RoboDK station: ICGI2018_station.rdk

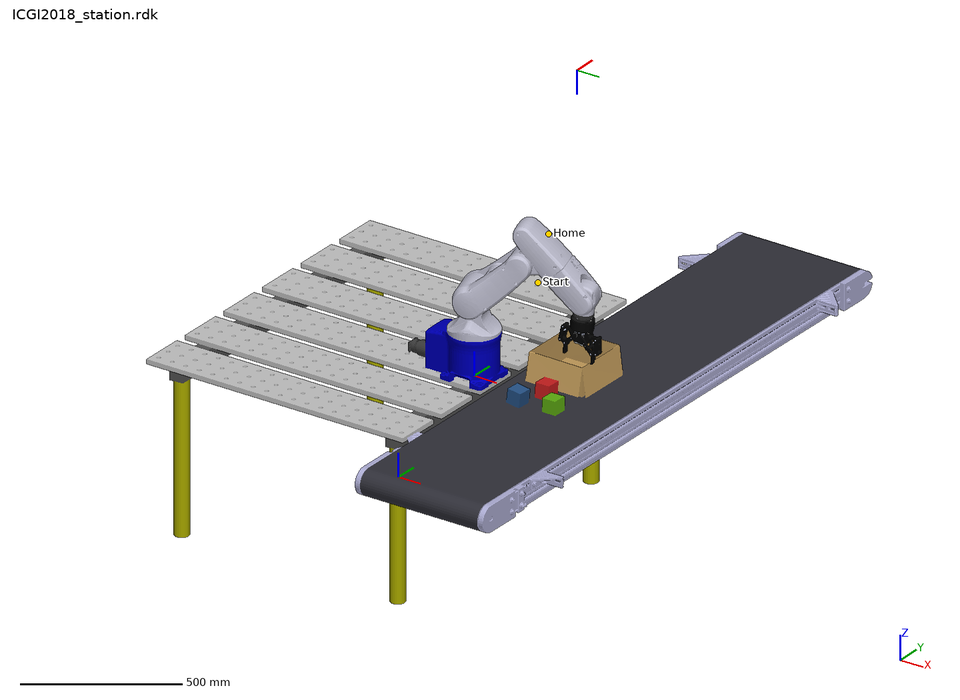
[picture v0: the station drawn from its stored meshes, robots at their saved joint values, targets as dots, program paths as lines]
Station ICGI2018_station. Poses are relative to the parent item; angles as X-Y-Z fixed-axis rotations.
  - frame ConveyorReference at (216.46, -62.53, 0) mm
    - object Conveyor at (-115.17, 300, -50) mm, size 597 x 2090.8 x 107.2 mm
    - object Opened Box at (-58.27, 786.37, -1) mm, size 224.8 x 231.5 x 101.8 mm, geometry from box.stl
  - object Object Table at (-409.94, 767.55, 0) mm, rotated rx 0 ry 0 rz -90.17 deg, size 1193.8 x 965.2 x 609.6 mm, geometry from Object Table.wrl
  - program ResetPositions (1 instructions, listed below)
  - frame Camera Frame at (325.51, 738.58, 1103.48) mm, rotated rx -180 ry 0 rz 90 deg
  - frame Denso VP-6242 Base at (0, 653.31, 0) mm
    - robot Denso VP-6242: 6 axes, payload 2 kg, reach 432 mm, repeatability 0.02 mm, weight 15 kg
        modified DH rows (alpha deg, a mm, theta deg, d mm): 0, 0, 0, 280; -90, 0, -90, 0; 0, 210, -90, 0; -90, 75, 0, 210; 90, 0, 0, 0; -90, 0, 0, 70
        joint limits [-160, -120, 19, -160, -120, -360] to [160, 120, 160, 160, 120, 360]; home [0, 0, 90, 0, 0, 0]; saved at [18.272, 48.672, 88.261, 2.665, 49.222, 16.423]
      - tool Gripper RobotiQ 85 Fully closed, TCP at (0, -20, 130) mm, size 121.5 x 160.2 x 75 mm
      - tool Gripper RobotiQ 85 Closed, TCP at (0, -20, 130) mm, size 134.4 x 157.6 x 75 mm
      - tool Gripper RobotiQ 85 Opened, TCP at (0, -20, 130) mm, size 147.4 x 146.8 x 75 mm
    - target Home (Cartesian target) at (280, 0, 565) mm, rotated rx 0 ry -90 rz -180 deg; joints [-14.036, -32.466, 113.204, 57.227, 16.765, -56.084] of Denso VP-6242
    - target Start (Cartesian target) at (240.34, 0, 387.41) mm, rotated rx -180 ry 6.45 rz 0 deg; joints [-4.352, 18.952, 61.872, -0.507, 105.605, -4.461] of Denso VP-6242
  - object Cube R at (267.82, 659.35, 26.94) mm, rotated rx -179.99 ry 1.92 rz 90.24 deg, size 51.6 x 51.6 x 51.6 mm, geometry from mini_box.stl
  - object Cube G at (338.43, 594.43, 20.96) mm, rotated rx 179.26 ry -0.01 rz 89.15 deg, size 50 x 50 x 50 mm, geometry from mini_box.stl
  - object Cube B at (221.28, 572.37, 26.97) mm, rotated rx -173.25 ry 0.31 rz 87.36 deg, size 50 x 50 x 50 mm, geometry from mini_box.stl

--- program ResetPositions ---
  Replace objects
